// TIA Portal V20 export
DATA_BLOCK "DB_MachineOptions"   // DB1300
{ S7_Optimized_Access := 'FALSE'; DB_Accessible_From_OPC_UA := 'FALSE' }
// stored: AutoNumber false, DBAccessibleFromOPCUA false, DBAccessibleFromWebserver false
   VAR RETAIN
      UPSPresent : Bool;
      Fixture : Struct
         Passive_Open : Bool;
      END_STRUCT;
      Mach_MONO_DUO : Bool;
      Chiller : Struct
         Termotek : Bool := TRUE;
         SMC : Bool := FALSE;
      END_STRUCT;
   END_VAR
BEGIN
END_DATA_BLOCK
